// TIA Portal V20 export
TYPE "LGM_LKinCtrl_ControlNode"
// stored: Access Published
   STRUCT
      commandConfiguration : "LGM_LKinCtrl_ControlNodeConfig";
      commands : "LGM_LKinCtrl_ControlNodeCommands";
      monitoring : "LGM_LKinCtrl_ControlNodeMonitoring";
   END_STRUCT;
   // monitoring.groupPower.diagnostics.status := 0;
END_TYPE
